// TIA Portal project "motore accelerazione-decelerazione" (V11)

(* hardware
DEVICE "Stazione SIMATIC 1200_1"  S71200.Device
   slot 0: "Telaio di montaggio S7-1200"  Rack  V1.0
   slot 1: "PLC_1"  CPU 1214C AC/DC/Rly  6ES7 214-1BE30-0XB0  V2.0
*)

// ===== PLC "PLC_1"  CPU 1214C AC/DC/Rly =====

VAR_GLOBAL   // PLC tag table "Tabella delle variabili standard"
   "Tag_1" AT %Q0.0 : Bool;
END_VAR

VAR_GLOBAL   // PLC tag table "Tabella delle variabili_1"
   "mw100" AT %MW100 : Int;
   "i0.0" AT %I0.1 : Bool;
   "qw80" AT %QW80 : Int;
   "md10" AT %MD10 : DInt;
END_VAR

// folder: System blocks/Program resources

DATA_BLOCK "tmr1"   // DB1
{ S7_Optimized_Access := 'FALSE' }
AUTHOR : Simatic
FAMILY : IEC
NAME : IEC_TMR
VERSION : 1.0
// stored: InstanceOfName ?
"?"
BEGIN
END_DATA_BLOCK

DATA_BLOCK "tmr2"   // DB2
{ S7_Optimized_Access := 'FALSE' }
AUTHOR : Simatic
FAMILY : IEC
NAME : IEC_TMR
VERSION : 1.0
// stored: InstanceOfName ?
"?"
BEGIN
END_DATA_BLOCK

DATA_BLOCK "IEC_Timer_0_DB"   // DB3
{ S7_Optimized_Access := 'FALSE' }
AUTHOR : Simatic
FAMILY : IEC
NAME : IEC_TMR
VERSION : 1.0
// stored: InstanceOfName ?
"?"
BEGIN
END_DATA_BLOCK

DATA_BLOCK "tmr3"   // DB4
{ S7_Optimized_Access := 'FALSE' }
AUTHOR : Simatic
FAMILY : IEC
NAME : IEC_TMR
VERSION : 1.0
// stored: InstanceOfName ?
"?"
BEGIN
END_DATA_BLOCK

// folder: (top level)

ORGANIZATION_BLOCK "Main"   // OB1, LAD, ProgramCycle
TITLE = "Main Program Sweep (Cycle)"
{ S7_Optimized_Access := 'FALSE' }
VERSION : 0.1
   VAR_TEMP   // added for the SCL form of the ladder/FBD networks
      _w1 : Bool;
   END_VAR
BEGIN

REGION Network 1
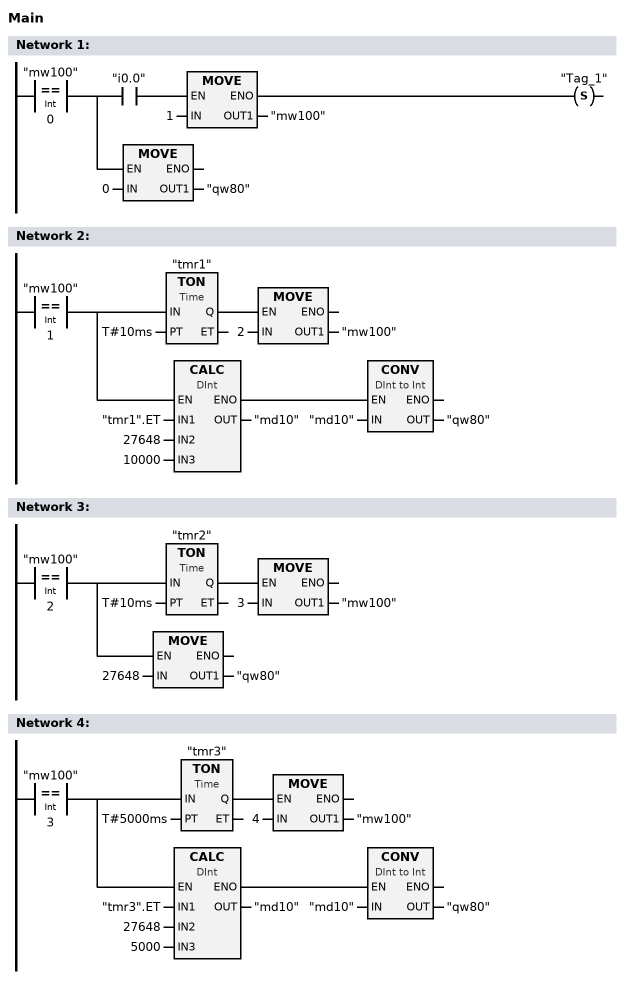
   RUNG wire#powerrail
      { S7_Templates := "SrcType := Int" } EQ_Contact(in1 := "mw100", in2 := 0)
      wire#w1
      Contact( "i0.0" )
      { S7_GenerateENO := "TRUE" } Move(in := 1, out1 => "mw100")
      S_Coil( "Tag_1" )
   END_RUNG
   RUNG wire#w1
      { S7_GenerateENO := "TRUE" } Move(in := 0, out1 => "qw80")
   END_RUNG
   // the same network as SCL:
   // ENO of a box is taken as its EN; it also drops when the box reports an error
   #_w1 := "mw100" = 0;
   IF #_w1 AND "i0.0" THEN
       "mw100" := 1;
       "Tag_1" := TRUE;
   END_IF;
   IF #_w1 THEN "qw80" := 0; END_IF;
END_REGION

REGION Network 2
   // ENO of a box is taken as its EN; it also drops when the box reports an error
   #_w1 := "mw100" = 1;
   "tmr1".TON(IN := #_w1, PT := T#10ms);
   IF "tmr1".Q THEN "mw100" := 2; END_IF;
   IF #_w1 THEN
       CALC(in1 := "tmr1".ET, in2 := 27648, in3 := 10000, out => "md10");
       "qw80" := DINT_TO_INT("md10");
   END_IF;
END_REGION

REGION Network 3
   #_w1 := "mw100" = 2;
   "tmr2".TON(IN := #_w1, PT := T#10ms);
   IF "tmr2".Q THEN "mw100" := 3; END_IF;
   IF #_w1 THEN "qw80" := 27648; END_IF;
END_REGION

REGION Network 4
   // ENO of a box is taken as its EN; it also drops when the box reports an error
   #_w1 := "mw100" = 3;
   "tmr3".TON(IN := #_w1, PT := T#5000ms);
   IF "tmr3".Q THEN "mw100" := 4; END_IF;
   IF #_w1 THEN
       CALC(in1 := "tmr3".ET, in2 := 27648, in3 := 5000, out => "md10");
       "qw80" := DINT_TO_INT("md10");
   END_IF;
END_REGION
END_ORGANIZATION_BLOCK